(* Schneider Machine Expert - Basic project automated warehouse lamp control, file version 2.7.0.0 *)
(* ProjectInformations: Name=New project *)

HARDWARE
  Cpu 0: TM221M16R/G
  EthernetConfiguration: NetworkName=M221, IpAllocationMode=FixedAddress, IpAddress=0.0.0.0, SubnetMask=0.0.0.0
  SerialLineConfiguration: Baud=Baud19200, Parity=ParityEven, DataBits=DataBits8, StopBits=StopBits1, PhysicalMedium=PhysicalMediumRs485, TransmissionMode=TransmissionModeModbusRtu, SlaveId=1, Addressing=SlaveAddressing
  MastTask: UsePeriodScanMode=false, PeriodScan=100
  FastTask: Period=255
  CpuBehavior: StartingMode=StartAsPreviousState, AutoSaveRamOnEeprom=true, WatchdogPeriod=250

SYMBOLS  (address, symbol, comment, settings)
  %M0       ON_OFF
  %I0.0     ENTER
  %I0.1     EXIT
  %I0.2     SECTION1
  %I0.3     SECTION2
  %I0.4     SECTION3
  %Q0.0     SECTION1_LAMP
  %Q0.1     SECTION2_LAMP
  %Q0.2     SECTION3_LAMP

POU New POU
  (* SectionNumber=0 *)

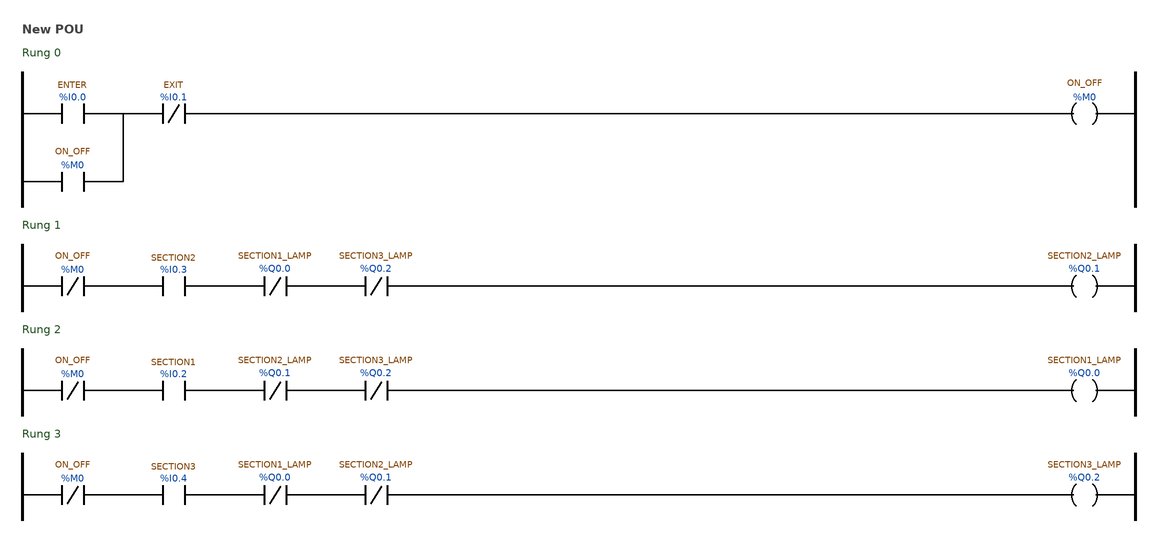

// Rung 0
  LD %I0.0                (* ENTER *)
  OR %M0                  (* ON_OFF *)
  ANDN %I0.1              (* EXIT *)
  ST %M0                  (* ON_OFF *)
  // as ST:
  //   ON_OFF := (ENTER OR ON_OFF) AND NOT EXIT;

// Rung 1
  LDN %M0                 (* ON_OFF *)
  AND %I0.3               (* SECTION2 *)
  ANDN %Q0.0              (* SECTION1_LAMP *)
  ANDN %Q0.2              (* SECTION3_LAMP *)
  ST %Q0.1                (* SECTION2_LAMP *)
  // as ST:
  //   SECTION2_LAMP := NOT ON_OFF AND SECTION2 AND NOT SECTION1_LAMP AND NOT SECTION3_LAMP;

// Rung 2
  LDN %M0                 (* ON_OFF *)
  AND %I0.2               (* SECTION1 *)
  ANDN %Q0.1              (* SECTION2_LAMP *)
  ANDN %Q0.2              (* SECTION3_LAMP *)
  ST %Q0.0                (* SECTION1_LAMP *)
  // as ST:
  //   SECTION1_LAMP := NOT ON_OFF AND SECTION1 AND NOT SECTION2_LAMP AND NOT SECTION3_LAMP;

// Rung 3
  LDN %M0                 (* ON_OFF *)
  AND %I0.4               (* SECTION3 *)
  ANDN %Q0.0              (* SECTION1_LAMP *)
  ANDN %Q0.1              (* SECTION2_LAMP *)
  ST %Q0.2                (* SECTION3_LAMP *)
  // as ST:
  //   SECTION3_LAMP := NOT ON_OFF AND SECTION3 AND NOT SECTION1_LAMP AND NOT SECTION2_LAMP;
